(*
    Tc2_System's F_GetSystemTime / F_GetTaskTime, supplied by
    samples/xStunit.SystemLibraryPlugins.

    The whole point is that neither reads wall time. A test that asked the
    machine what time it is could assert nothing at all - it would pass here
    and fail on a different machine, or a second later. These read the
    interpreter's simulated clock instead, so AdvanceClock moves them by
    exactly what it says and an absolute timestamp is a constant a test can
    write down.

    125911584000000000 is 2000-01-01T00:00:00Z in the vendor's unit: 100 ns
    intervals since 1601-01-01 UTC, which is the epoch both functions answer
    in and is also where the simulated clock's origin sits.

    The clock is shared by every suite in a RUN, not just a file, and there is
    no ST way to set it back. That is why this suite sits in a fixture
    directory of its own: the absolute assertion below needs the clock to still
    be at its origin, and any suite sharing the run that advanced it first -
    the ADS timeout test does exactly that - would move the answer.
*)
FUNCTION_BLOCK FB_TimePluginTests EXTENDS TcUnit.FB_TestSuite

SystemTimeStartsAtTheSimulatedOrigin();
SystemTimeFollowsTheSimulatedClock();
TaskTimeStaysAtTheStartOfTheCycle();

METHOD PRIVATE SystemTimeStartsAtTheSimulatedOrigin
VAR
	tNow		: ULINT;
END_VAR
TEST('SystemTimeStartsAtTheSimulatedOrigin');

tNow := F_GetSystemTime();

(* An absolute constant, which is only writable at all because the clock is
   simulated. This also pins the epoch: a function counting from 1970 rather
   than 1601 would be out by 369 years here. *)
AssertEquals_ULINT(Expected := 125911584000000000,
                    Actual := tNow,
                    Message := 'system time starts at the simulated origin');

TEST_FINISHED();
END_METHOD

METHOD PRIVATE SystemTimeFollowsTheSimulatedClock
VAR
	tBefore		: ULINT;
	tAfter		: ULINT;
END_VAR
TEST('SystemTimeFollowsTheSimulatedClock');

tBefore := F_GetSystemTime();
AdvanceClock(T#500MS);
tAfter := F_GetSystemTime();

(* 500 ms is 5 000 000 units of 100 ns. A function reading wall time would
   report an arbitrary difference here instead. *)
AssertEquals_ULINT(Expected := 5000000,
                    Actual := tAfter - tBefore,
                    Message := 'the clock advance is exactly what system time moved by');

TEST_FINISHED();
END_METHOD

METHOD PRIVATE TaskTimeStaysAtTheStartOfTheCycle
VAR
	tTask		: ULINT;
	tTaskAgain	: ULINT;
	tSystem		: ULINT;
END_VAR
TEST('TaskTimeStaysAtTheStartOfTheCycle');

tTask := F_GetTaskTime();
AdvanceClock(T#250MS);
tTaskAgain := F_GetTaskTime();
tSystem := F_GetSystemTime();

(* The documented difference between the two: a task's start time does not
   move part-way through its own cycle, so two reads in one cycle agree even
   though system time has moved between them. *)
AssertEquals_ULINT(Expected := tTask,
                    Actual := tTaskAgain,
                    Message := 'task time does not move within a cycle');
AssertEquals_BOOL(Expected := TRUE,
                   Actual := tSystem > tTaskAgain,
                   Message := 'system time did move within the same cycle');

TEST_FINISHED();
END_METHOD

END_FUNCTION_BLOCK

(* stored: Version 1.1.0.1, ProductVersion 3.1.4026.18
   POU FB_TimePluginTests: Id {b2c3d4e5-6k20-4a1a-8b1b-000000000030}, SpecialFunc None
   Method SystemTimeStartsAtTheSimulatedOrigin: Id {b2c3d4e5-6k20-4a1a-8b1b-000000000031}
   Method SystemTimeFollowsTheSimulatedClock: Id {b2c3d4e5-6k20-4a1a-8b1b-000000000032}
   Method TaskTimeStaysAtTheStartOfTheCycle: Id {b2c3d4e5-6k20-4a1a-8b1b-000000000033} *)
